{attribute 'pack_mode' := '1'}
TYPE ST_AdsLogStringMessage :
STRUCT
	MsgCtrlMask : DWORD;
    MsgFmtStr : Tc2_System.T_MaxString;
    StrArg : Tc2_System.T_MaxString;
END_STRUCT
END_TYPE

(* stored: Version 1.1.0.1
   DUT ST_AdsLogStringMessage: Id {7eac3ec2-a59e-45fa-bfc5-ba06a20b9608} *)
